PROGRAM POU_Output
VAR
END_VAR
//tower Lamp POU

// NETWORK 1

END_PROGRAM

(* stored: Version 1.1.0.1, ProductVersion 3.1.4024.0
   POU POU_Output: Id {e8319bc5-7c65-4ad5-898d-7dcfb385da92}, SpecialFunc None *)
